FUNCTION_BLOCK FB_ErrorHandler_abond EXTENDS FB_ActionBasic
VAR_INPUT
	xEnable : BOOL;
	stAdmin : REFERENCE TO ST_PMLa;
	AlarmList :REFERENCE TO ARRAY[0..999] OF ST_Alarm_Tmax;
END_VAR
VAR_OUTPUT
END_VAR
VAR
	StateBehavior : CBML.LConC;
	ErrorCount : DINT;
END_VAR

THIS^.IBehaviourModel := StateBehavior;
StateBehavior(xEnable:= xEnable, xBusy=> xBusy, xError=> xError);
//AlarmCtrl();
//IF btest THEN
//stAlarm.Trigger := TRUE;
//stAlarm.Message := 'test';
//AlarmCtrl.M_SetAlarm(stAdmin := GVL_Machine.PackTags[0].Admin, stAlarm := stAlarm);
//END_IF

METHOD CleanupAction
VAR_INPUT
    xAbortProposed : BOOL;
    iErrorIDProposed: INT;
END_VAR
VAR_OUTPUT
    xComplete : BOOL := TRUE;
    xAbort: BOOL := xAbortProposed;
 	iErrorID : INT := iErrorIDProposed;
END_VAR
END_METHOD

METHOD CyclicAction
VAR_INPUT
    itfTimingController : CBML.ITimingController;
END_VAR
VAR_OUTPUT
    xComplete : BOOL := TRUE;
    iErrorID : INT := 0;
END_VAR
VAR
	diCheckTriggerLoop : DINT;
	diCheckAlarmLoop : DINT;
	bHasSameID :BOOL;
END_VAR
VAR_INST
	diSearchID : DINT;
END_VAR
xComplete := FALSE;
bHasSameID := FALSE;
diSearchID := 0;
FOR diCheckTriggerLoop := 1 TO stAdmin.AlarmExtent DO
    IF stAdmin.Alarm[diCheckTriggerLoop].Trigger THEN
        FOR diCheckAlarmLoop := 0 TO 999 DO
            IF AlarmList[diCheckAlarmLoop].ID = stAdmin.Alarm[diCheckTriggerLoop].ID THEN
				diSearchID := diCheckTriggerLoop;
                bHasSameID := TRUE;
				EXIT;
            END_IF
        END_FOR
    END_IF

    IF NOT bHasSameID THEN
        ErrorCount := ErrorCount + 1;
        AlarmList[ErrorCount].ID := DINT_TO_UDINT(stAdmin.Alarm[diCheckTriggerLoop].ID);
        AlarmList[ErrorCount].Category := stAdmin.Alarm[diCheckTriggerLoop].Category;
        AlarmList[ErrorCount].Message := stAdmin.Alarm[diCheckTriggerLoop].Message;
        AlarmList[ErrorCount].Value := stAdmin.Alarm[diCheckTriggerLoop].Value;
        AlarmList[ErrorCount].Trigger := stAdmin.Alarm[diCheckTriggerLoop].Trigger;
    END_IF
END_FOR
END_METHOD

METHOD ExitAction
VAR_INPUT
    xAfterCleanup : BOOL;
    xInCopyCode : BOOL;
END_VAR
END_METHOD

METHOD ResetAction
VAR_OUTPUT
    xComplete : BOOL := TRUE;
END_VAR
END_METHOD

METHOD StartAction
VAR_OUTPUT
    xComplete : BOOL := TRUE;
	iErrorID : INT := 0;
END_VAR
END_METHOD

END_FUNCTION_BLOCK

(* stored: Version 1.1.0.1, ProductVersion 3.1.4024.13
   POU FB_ErrorHandler_abond: Id {e31cc1cf-3e71-4ee6-a485-d500ce5c0dad}, SpecialFunc None
   Method CleanupAction: Id {e2b56292-7be8-49f6-8fb6-50485b35f384}
   Method CyclicAction: Id {6f06e8e0-bb95-40e8-961f-04ccc872cb0e}
   Method ExitAction: Id {3e89ca1a-665d-4a55-8d6f-a20bc678ed61}
   Method ResetAction: Id {28e35ddc-0c9f-4a1a-b51b-2748d058b758}
   Method StartAction: Id {14f4669e-e1a8-4f0a-b23e-f7f51b01b19f} *)
